{attribute 'pack_mode' := '2'}
TYPE ST_MOTION_FUNCTION :
STRUCT
  stMotionFunction            : ARRAY[1..MAX_MOTION_FUNCTION_POINTS] OF ST_MOTION_FUNCTION_POINT;
  nMotionFunctionSize         : UINT;
  nPoints                     : UINT; // number of points used in motion function 
END_STRUCT
END_TYPE

(* stored: Version 1.1.0.1
   DUT ST_MOTION_FUNCTION: Id {bf9669c6-cca8-4a6d-b300-a9aaf781c877} *)
